FUNCTION_BLOCK MONGO_DB_INSERT
  {SET_ATTRIBUTE(OpcUa, SERVICE)}
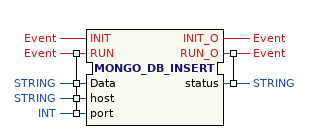
  EVENT_INPUT
    INIT;
    RUN WITH Data, host, port; {SET_ATTRIBUTE(OpcUa, Method)}
  END_EVENT
  EVENT_OUTPUT
    INIT_O;
    RUN_O WITH status;
  END_EVENT
  VAR_INPUT
    Data : STRING; {SET_ATTRIBUTE(OpcUa, Variable.RUN)}
    host : STRING; {SET_ATTRIBUTE(OpcUa, Variable.RUN)}
    port : INT; {SET_ATTRIBUTE(OpcUa, Variable.RUN)}
  END_VAR
  VAR_OUTPUT
    status : STRING; {SET_ATTRIBUTE(OpcUa, Variable.RUN)}
  END_VAR
END_FUNCTION_BLOCK
